Yaskawa INFORM job: driller_case_upwards_cylinder_program.JBI

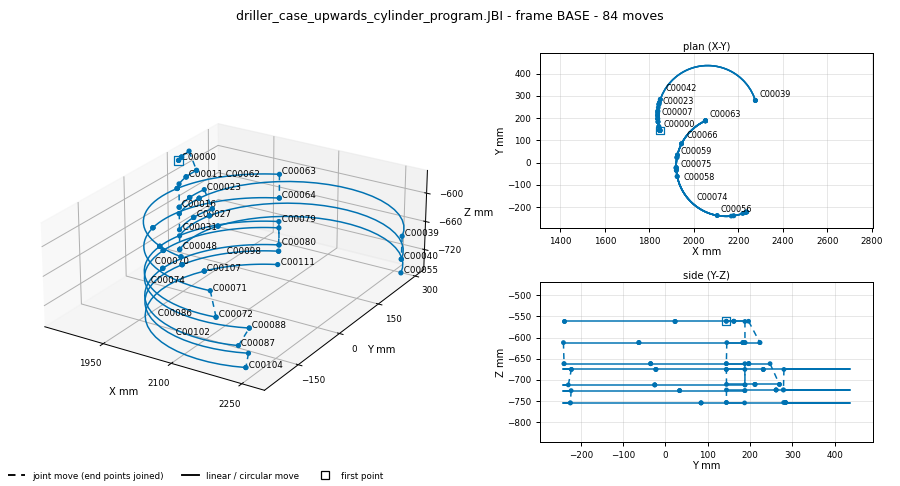
[picture p0: tool path of driller_case_upwards_cylinder_program.JBI in frame BASE, 84 of 117 moves have a stored position in this frame; points joined in program order, loops and branches not executed]
/JOB
//NAME driller_case_upwards_cylinder_program
//POS
///NPOS 112,0,112,0,0,0
///TOOL 0
///POSTYPE BASE
///RECTAN
///RCONF 0,0,0,0,0,0,0,0,0,0,0,0,0,0,0,0,0,0,0,0,0,0,0,0
C00000=1847.483471,143.792175,-561.434000,-162.596187,-90.000000,5.000000
C00001=1847.483471,143.792175,-561.434000,-162.596187,-90.000000,5.000000
C00002=1844.331938,154.825241,-561.434000,-165.520432,-90.000000,5.000000
C00003=1842.717405,161.496365,-561.434000,-167.269532,-90.000000,5.000000
C00004=1842.717405,161.496365,-561.434000,-167.269532,-90.000000,5.000000
C00005=1842.717405,161.496365,-561.434000,-167.269532,-90.000000,5.000000
C00006=1839.611038,178.138573,-561.434000,-171.584610,-90.000000,5.000000
C00007=1837.671696,196.336618,-561.434000,-175.000000,-89.999999,5.000000
C00008=1837.511507,223.061616,-611.872500,175.000000,-90.000000,5.000000
C00009=1837.511507,223.061616,-611.872500,175.000000,-90.000000,5.000000
C00010=1837.683187,196.162364,-611.872500,-175.000000,-89.999999,5.000000
C00011=1838.946943,182.992119,-611.872500,-172.832953,-90.000000,5.000000
C00012=1838.946943,182.992119,-611.872500,-172.832953,-90.000000,5.000000
C00013=1838.946943,182.992119,-611.872500,-172.832953,-90.000000,5.000000
C00014=1841.227991,168.624137,-611.872500,-169.125162,-89.999999,5.000000
C00015=1847.151839,144.859452,-611.872500,-162.880981,-90.000000,5.000000
C00016=1847.458309,143.872499,-661.563500,-162.617636,-90.000000,5.000000
C00017=1847.458309,143.872499,-661.563500,-162.617636,-90.000000,5.000000
C00018=1840.747860,171.204531,-661.563500,-169.793996,-90.000000,5.000000
C00019=1837.641591,196.803296,-661.563500,-175.000000,-89.999999,5.000000
C00020=1837.641591,196.803296,-661.563500,-175.000000,-89.999999,5.000000
C00021=1837.641591,196.803296,-661.563500,-175.000000,-89.999999,5.000000
C00022=1837.544765,223.667671,-661.563500,175.000000,-89.999999,5.000000
C00023=1840.087961,247.026739,-661.563500,170.791289,-90.000000,5.000000
C00024=1844.835805,269.179881,-710.495000,165.015523,-89.999999,5.000000
C00025=1844.835805,269.179881,-710.495000,165.015523,-89.999999,5.000000
C00026=1838.661141,236.721897,-710.495000,173.442487,-89.999999,5.000000
C00027=1837.190484,211.438050,-710.495000,175.000000,-90.000000,5.000000
C00028=1837.190484,211.438050,-710.495000,175.000000,-90.000000,5.000000
C00029=1837.190484,211.438050,-710.495000,175.000000,-90.000000,5.000000
C00030=1838.560307,186.259867,-710.495000,-173.671466,-90.000000,5.000000
C00031=1847.367305,144.163901,-710.495000,-162.695429,-90.000000,5.000000
C00032=1847.465652,143.849049,-675.202960,175.000000,-60.000000,17.388625
C00033=1847.465652,143.849049,-675.202960,175.000000,-60.000000,17.388625
C00034=1838.198632,189.772547,-675.202960,175.000000,-60.000000,5.428681
C00035=1838.082959,231.061815,-675.202960,175.000000,-60.000000,-5.107650
C00036=1838.082959,231.061815,-675.202960,175.000000,-60.000000,-5.107650
C00037=1838.082959,231.061815,-675.202960,175.000000,-60.000000,-5.107650
C00038=1843.291277,263.067526,-675.202960,175.000000,-60.000000,-13.377898
C00039=2276.120949,279.768364,-675.202960,-175.000000,-60.000000,-162.202751
C00040=2276.486372,278.619440,-723.587460,175.000000,-60.000000,-162.509975
C00041=2276.486372,278.619440,-723.587460,175.000000,-60.000000,-162.509975
C00042=1856.876158,303.050330,-723.587460,175.000000,-60.000000,-24.154345
C00043=1842.881938,261.315233,-723.587460,-175.000000,-60.000000,-12.919351
C00044=1842.881938,261.315233,-723.587460,-175.000000,-60.000000,-12.919351
C00045=1842.881938,261.315233,-723.587460,-175.000000,-60.000000,-12.919351
C00046=1837.219332,214.667491,-723.587460,175.000000,-60.000000,-5.000000
C00047=1847.384163,144.109815,-723.587460,-175.000000,-60.000000,17.319007
C00048=1847.444853,143.915500,-753.280960,-175.000000,-60.000000,17.370882
C00049=1847.444853,143.915500,-753.280960,-175.000000,-60.000000,17.370882
C00050=1837.847810,228.229189,-753.280960,-175.000000,-60.000000,-5.000000
C00051=1849.201992,283.551928,-753.280960,175.000000,-60.000000,-18.812789
C00052=1849.201992,283.551928,-753.280960,175.000000,-60.000000,-18.812789
C00053=1849.201992,283.551928,-753.280960,175.000000,-60.000000,-18.812789
C00054=2263.742893,310.390706,-753.280960,175.000000,-60.000000,-153.778507
C00055=2276.298981,279.211279,-753.280960,-175.000000,-60.000000,-162.351782
C00056=2104.976134,-238.300239,-561.969000,-100.335590,-89.999999,5.000000
C00057=2104.976134,-238.300239,-561.969000,-100.335590,-89.999999,5.000000
C00058=1934.437143,-95.112312,-561.969000,-159.699386,-90.000000,5.000000
C00059=1924.039557,22.797395,-561.969000,169.778297,-90.000000,5.000000
C00060=1924.039557,22.797395,-561.969000,169.778297,-90.000000,5.000000
C00061=1924.039557,22.797395,-561.969000,169.778297,-90.000000,5.000000
C00062=1967.007068,119.868678,-561.969000,142.469628,-90.000000,5.000000
C00063=2052.547133,187.712297,-561.969000,114.367716,-90.000000,5.000000
C00064=2052.634052,187.751645,-611.842000,114.343403,-89.999999,5.000000
C00065=2052.634052,187.751645,-611.842000,114.343403,-89.999999,5.000000
C00066=1948.511703,91.632351,-611.842000,151.079153,-89.999999,5.000000
C00067=1925.136531,-62.669770,-611.842000,-168.307591,-90.000000,5.000000
C00068=1925.136531,-62.669770,-611.842000,-168.307591,-90.000000,5.000000
C00069=1925.136531,-62.669770,-611.842000,-168.307591,-90.000000,5.000000
C00070=2016.668432,-201.508108,-611.842000,-124.901105,-90.000000,5.000000
C00071=2168.016110,-240.799851,-611.842000,-84.205726,-90.000000,5.000000
C00072=2178.982831,-239.413884,-661.628500,-81.388642,-89.999999,5.000000
C00073=2178.982831,-239.413884,-661.628500,-81.388642,-89.999999,5.000000
C00074=1996.690438,-185.821293,-661.628500,-131.377236,-90.000000,5.000000
C00075=1921.175947,-34.895000,-661.628500,-175.000000,-90.000000,5.000000
C00076=1921.175947,-34.895000,-661.628500,-175.000000,-90.000000,5.000000
C00077=1921.175947,-34.895000,-661.628500,-175.000000,-90.000000,5.000000
C00078=1938.754866,71.710304,-661.628500,156.734175,-89.999999,5.000000
C00079=2052.189521,187.549944,-661.628500,114.467795,-90.000000,5.000000
C00080=2052.696354,187.779820,-711.669000,114.325979,-90.000000,5.000000
C00081=2052.696354,187.779820,-711.669000,114.325979,-90.000000,5.000000
C00082=1950.004096,94.290755,-711.669000,150.302278,-90.000000,5.000000
C00083=1920.617518,-25.221347,-711.669000,-175.000000,-90.000000,5.000000
C00084=1920.617518,-25.221347,-711.669000,-175.000000,-90.000000,5.000000
C00085=1920.617518,-25.221347,-711.669000,-175.000000,-90.000000,5.000000
C00086=2026.210016,-207.810144,-711.669000,-121.986910,-90.000000,5.000000
C00087=2219.589727,-229.327007,-711.669000,-70.711167,-89.999999,5.000000
C00088=2237.806700,-222.044697,-675.142960,175.000000,-60.000000,114.289693
C00089=2237.806700,-222.044697,-675.142960,175.000000,-60.000000,114.289693
C00090=2092.243379,-235.595126,-675.142960,-175.000000,-60.000000,76.346933
C00091=1920.536336,-22.526760,-675.142960,-175.000000,-60.000000,5.000000
C00092=1920.536336,-22.526760,-675.142960,-175.000000,-60.000000,5.000000
C00093=1920.536336,-22.526760,-675.142960,-175.000000,-60.000000,5.000000
C00094=1955.704025,103.738259,-675.142960,-175.000000,-60.000000,-32.509666
C00095=2052.244332,187.574877,-675.142960,175.000000,-60.000000,-65.547549
C00096=2052.113028,187.515119,-725.239460,175.000000,-60.000000,-65.510788
C00097=2052.113028,187.515119,-725.239460,175.000000,-60.000000,-65.510788
C00098=1967.085350,119.970526,-725.239460,-175.000000,-60.000000,-37.563106
C00099=1926.239510,33.501310,-725.239460,175.000000,-60.000000,-13.006593
C00100=1926.239510,33.501310,-725.239460,175.000000,-60.000000,-13.006593
C00101=1926.239510,33.501310,-725.239460,175.000000,-60.000000,-13.006593
C00102=2082.559050,-233.012862,-725.239460,-175.000000,-60.000000,73.792711
C00103=2236.529777,-222.616199,-725.239460,-175.000000,-60.000000,113.933200
C00104=2232.212846,-224.478415,-754.172960,-175.000000,-60.000000,112.735139
C00105=2232.212846,-224.478415,-754.172960,-175.000000,-60.000000,112.735139
C00106=1923.080705,17.055163,-754.172960,175.000000,-60.000000,-8.738149
C00107=1944.567746,84.166172,-754.172960,-175.000000,-60.000000,-26.769034
C00108=1944.567746,84.166172,-754.172960,-175.000000,-60.000000,-26.769034
C00109=1944.567746,84.166172,-754.172960,-175.000000,-60.000000,-26.769034
C00110=1980.831204,136.194342,-754.172960,175.000000,-60.000000,-42.983699
C00111=2050.689223,186.860577,-754.172960,-175.000000,-60.000000,-65.111467
///POSTYPE PULSE
///PULSE
EX00000=17408.0
EX00001=301056.0
///POSTYPE PULSE
///PULSE
EC00000=17408.0
EC00001=17408.0
EC00002=17408.0
EC00003=17408.0
EC00004=17408.0
EC00005=17408.0
EC00006=17408.0
EC00007=17408.0
EC00008=17408.0
EC00009=17408.0
EC00010=17408.0
EC00011=17408.0
EC00012=17408.0
EC00013=17408.0
EC00014=17408.0
EC00015=17408.0
EC00016=17408.0
EC00017=17408.0
EC00018=17408.0
EC00019=17408.0
EC00020=17408.0
EC00021=17408.0
EC00022=17408.0
EC00023=17408.0
EC00024=17408.0
EC00025=17408.0
EC00026=17408.0
EC00027=17408.0
EC00028=17408.0
EC00029=17408.0
EC00030=17408.0
EC00031=17408.0
EC00032=17408.0
EC00033=17408.0
EC00034=17408.0
EC00035=17408.0
EC00036=17408.0
EC00037=17408.0
EC00038=17408.0
EC00039=17408.0
EC00040=17408.0
EC00041=17408.0
EC00042=17408.0
EC00043=17408.0
EC00044=17408.0
EC00045=17408.0
EC00046=17408.0
EC00047=17408.0
EC00048=17408.0
EC00049=17408.0
EC00050=17408.0
EC00051=17408.0
EC00052=17408.0
EC00053=17408.0
EC00054=17408.0
EC00055=17408.0
EC00056=301056.0
EC00057=301056.0
EC00058=301056.0
EC00059=301056.0
EC00060=301056.0
EC00061=301056.0
EC00062=301056.0
EC00063=301056.0
EC00064=301056.0
EC00065=301056.0
EC00066=301056.0
EC00067=301056.0
EC00068=301056.0
EC00069=301056.0
EC00070=301056.0
EC00071=301056.0
EC00072=301056.0
EC00073=301056.0
EC00074=301056.0
EC00075=301056.0
EC00076=301056.0
EC00077=301056.0
EC00078=301056.0
EC00079=301056.0
EC00080=301056.0
EC00081=301056.0
EC00082=301056.0
EC00083=301056.0
EC00084=301056.0
EC00085=301056.0
EC00086=301056.0
EC00087=301056.0
EC00088=301056.0
EC00089=301056.0
EC00090=301056.0
EC00091=301056.0
EC00092=301056.0
EC00093=301056.0
EC00094=301056.0
EC00095=301056.0
EC00096=301056.0
EC00097=301056.0
EC00098=301056.0
EC00099=301056.0
EC00100=301056.0
EC00101=301056.0
EC00102=301056.0
EC00103=301056.0
EC00104=301056.0
EC00105=301056.0
EC00106=301056.0
EC00107=301056.0
EC00108=301056.0
EC00109=301056.0
EC00110=301056.0
EC00111=301056.0
//INST
///DATE 2023/08/04 15:15
///ATTR SC,RW,RJ
////FRAME BASE
///GROUP1 RB1,ST1
NOP
MOVJ P009 EX000 VJ=15.00
MOVJ C00000 EC00000 VJ=15.0
CALL JOB:SPYON
MOVC C00001 EC00001 V=150.0
MOVC C00002 EC00002 V=150.0
MOVC C00003 EC00003 V=150.0
MOVJ C00004 EC00004 VJ=15.0
MOVC C00005 EC00005 V=150.0
MOVC C00006 EC00006 V=150.0
MOVC C00007 EC00007 V=150.0
MOVJ C00008 EC00008 VJ=15.0
MOVC C00009 EC00009 V=150.0
MOVC C00010 EC00010 V=150.0
MOVC C00011 EC00011 V=150.0
MOVJ C00012 EC00012 VJ=15.0
MOVC C00013 EC00013 V=150.0
MOVC C00014 EC00014 V=150.0
MOVC C00015 EC00015 V=150.0
MOVJ C00016 EC00016 VJ=15.0
MOVC C00017 EC00017 V=150.0
MOVC C00018 EC00018 V=150.0
MOVC C00019 EC00019 V=150.0
MOVJ C00020 EC00020 VJ=15.0
MOVC C00021 EC00021 V=150.0
MOVC C00022 EC00022 V=150.0
MOVC C00023 EC00023 V=150.0
MOVJ C00024 EC00024 VJ=15.0
MOVC C00025 EC00025 V=150.0
MOVC C00026 EC00026 V=150.0
MOVC C00027 EC00027 V=150.0
MOVJ C00028 EC00028 VJ=15.0
MOVC C00029 EC00029 V=150.0
MOVC C00030 EC00030 V=150.0
MOVC C00031 EC00031 V=150.0
MOVJ C00032 EC00032 VJ=15.0
MOVC C00033 EC00033 V=150.0
MOVC C00034 EC00034 V=150.0
MOVC C00035 EC00035 V=150.0
MOVJ C00036 EC00036 VJ=15.0
MOVC C00037 EC00037 V=150.0
MOVC C00038 EC00038 V=150.0
MOVC C00039 EC00039 V=150.0
MOVJ C00040 EC00040 VJ=15.0
MOVC C00041 EC00041 V=150.0
MOVC C00042 EC00042 V=150.0
MOVC C00043 EC00043 V=150.0
MOVJ C00044 EC00044 VJ=15.0
MOVC C00045 EC00045 V=150.0
MOVC C00046 EC00046 V=150.0
MOVC C00047 EC00047 V=150.0
MOVJ C00048 EC00048 VJ=15.0
MOVC C00049 EC00049 V=150.0
MOVC C00050 EC00050 V=150.0
MOVC C00051 EC00051 V=150.0
MOVJ C00052 EC00052 VJ=15.0
MOVC C00053 EC00053 V=150.0
MOVC C00054 EC00054 V=150.0
MOVC C00055 EC00055 V=150.0
CALL JOB:SPYOF
MOVJ P009 VJ=15.00
MOVL P009 EX00000 V=150.0
MOVJ C00056 EC00056 VJ=15.0
CALL JOB:SPYON
MOVC C00057 EC00057 V=150.0
MOVC C00058 EC00058 V=150.0
MOVC C00059 EC00059 V=150.0
MOVJ C00060 EC00060 VJ=15.0
MOVC C00061 EC00061 V=150.0
MOVC C00062 EC00062 V=150.0
MOVC C00063 EC00063 V=150.0
MOVJ C00064 EC00064 VJ=15.0
MOVC C00065 EC00065 V=150.0
MOVC C00066 EC00066 V=150.0
MOVC C00067 EC00067 V=150.0
MOVJ C00068 EC00068 VJ=15.0
MOVC C00069 EC00069 V=150.0
MOVC C00070 EC00070 V=150.0
MOVC C00071 EC00071 V=150.0
MOVJ C00072 EC00072 VJ=15.0
MOVC C00073 EC00073 V=150.0
MOVC C00074 EC00074 V=150.0
MOVC C00075 EC00075 V=150.0
MOVJ C00076 EC00076 VJ=15.0
MOVC C00077 EC00077 V=150.0
MOVC C00078 EC00078 V=150.0
MOVC C00079 EC00079 V=150.0
MOVJ C00080 EC00080 VJ=15.0
MOVC C00081 EC00081 V=150.0
MOVC C00082 EC00082 V=150.0
MOVC C00083 EC00083 V=150.0
MOVJ C00084 EC00084 VJ=15.0
MOVC C00085 EC00085 V=150.0
MOVC C00086 EC00086 V=150.0
MOVC C00087 EC00087 V=150.0
MOVJ C00088 EC00088 VJ=15.0
MOVC C00089 EC00089 V=150.0
MOVC C00090 EC00090 V=150.0
MOVC C00091 EC00091 V=150.0
MOVJ C00092 EC00092 VJ=15.0
MOVC C00093 EC00093 V=150.0
MOVC C00094 EC00094 V=150.0
MOVC C00095 EC00095 V=150.0
MOVJ C00096 EC00096 VJ=15.0
MOVC C00097 EC00097 V=150.0
MOVC C00098 EC00098 V=150.0
MOVC C00099 EC00099 V=150.0
MOVJ C00100 EC00100 VJ=15.0
MOVC C00101 EC00101 V=150.0
MOVC C00102 EC00102 V=150.0
MOVC C00103 EC00103 V=150.0
MOVJ C00104 EC00104 VJ=15.0
MOVC C00105 EC00105 V=150.0
MOVC C00106 EC00106 V=150.0
MOVC C00107 EC00107 V=150.0
MOVJ C00108 EC00108 VJ=15.0
MOVC C00109 EC00109 V=150.0
MOVC C00110 EC00110 V=150.0
MOVC C00111 EC00111 V=150.0
CALL JOB:SPYOF
MOVJ P009 VJ=15.00
MOVL P009 EX00001 V=150.0
END
